D11017	WORD	Память для хранения названий рецептов. Задание 41. Символ 18
D11018	WORD	Память для хранения названий рецептов. Задание 41. Символ 19
D11019	WORD	Память для хранения названий рецептов. Задание 41. Символ 20
D11020	WORD	Память для хранения названий рецептов. Задание 41. Символ 21
D11021	WORD	Память для хранения названий рецептов. Задание 41. Символ 22
D11022	WORD	Память для хранения названий рецептов. Задание 41. Символ 23
D11023	WORD	Память для хранения названий рецептов. Задание 41. Символ 24
D11024	WORD	Память для хранения названий рецептов. Задание 41. Символ 25
D11025	WORD	Память для хранения названий рецептов. Задание 42. Символ 1
D11026	WORD	Память для хранения названий рецептов. Задание 42. Символ 2
D11027	WORD	Память для хранения названий рецептов. Задание 42. Символ 3
D11028	WORD	Память для хранения названий рецептов. Задание 42. Символ 4
D11029	WORD	Память для хранения названий рецептов. Задание 42. Символ 5
D11030	WORD	Память для хранения названий рецептов. Задание 42. Символ 6
D11031	WORD	Память для хранения названий рецептов. Задание 42. Символ 7
D11032	WORD	Память для хранения названий рецептов. Задание 42. Символ 8
D11033	WORD	Память для хранения названий рецептов. Задание 42. Символ 9
D11034	WORD	Память для хранения названий рецептов. Задание 42. Символ 10
D11035	WORD	Память для хранения названий рецептов. Задание 42. Символ 11
D11036	WORD	Память для хранения названий рецептов. Задание 42. Символ 12
D11037	WORD	Память для хранения названий рецептов. Задание 42. Символ 13
D11038	WORD	Память для хранения названий рецептов. Задание 42. Символ 14
D11039	WORD	Память для хранения названий рецептов. Задание 42. Символ 15
D11040	WORD	Память для хранения названий рецептов. Задание 42. Символ 16
D11041	WORD	Память для хранения названий рецептов. Задание 42. Символ 17
D11042	WORD	Память для хранения названий рецептов. Задание 42. Символ 18
D11043	WORD	Память для хранения названий рецептов. Задание 42. Символ 19
D11044	WORD	Память для хранения названий рецептов. Задание 42. Символ 20
D11045	WORD	Память для хранения названий рецептов. Задание 42. Символ 21
D11046	WORD	Память для хранения названий рецептов. Задание 42. Символ 22
D11047	WORD	Память для хранения названий рецептов. Задание 42. Символ 23
D11048	WORD	Память для хранения названий рецептов. Задание 42. Символ 24
D11049	WORD	Память для хранения названий рецептов. Задание 42. Символ 25
D11050	WORD	Память для хранения названий рецептов. Задание 43. Символ 1
D11051	WORD	Память для хранения названий рецептов. Задание 43. Символ 2
D11052	WORD	Память для хранения названий рецептов. Задание 43. Символ 3
D11053	WORD	Память для хранения названий рецептов. Задание 43. Символ 4
D11054	WORD	Память для хранения названий рецептов. Задание 43. Символ 5
D11055	WORD	Память для хранения названий рецептов. Задание 43. Символ 6
D11056	WORD	Память для хранения названий рецептов. Задание 43. Символ 7
D11057	WORD	Память для хранения названий рецептов. Задание 43. Символ 8
D11058	WORD	Память для хранения названий рецептов. Задание 43. Символ 9
D11059	WORD	Память для хранения названий рецептов. Задание 43. Символ 10
D11060	WORD	Память для хранения названий рецептов. Задание 43. Символ 11
D11061	WORD	Память для хранения названий рецептов. Задание 43. Символ 12
D11062	WORD	Память для хранения названий рецептов. Задание 43. Символ 13
D11063	WORD	Память для хранения названий рецептов. Задание 43. Символ 14
D11064	WORD	Память для хранения названий рецептов. Задание 43. Символ 15
D11065	WORD	Память для хранения названий рецептов. Задание 43. Символ 16
D11066	WORD	Память для хранения названий рецептов. Задание 43. Символ 17
D11067	WORD	Память для хранения названий рецептов. Задание 43. Символ 18
D11068	WORD	Память для хранения названий рецептов. Задание 43. Символ 19
D11069	WORD	Память для хранения названий рецептов. Задание 43. Символ 20
D11070	WORD	Память для хранения названий рецептов. Задание 43. Символ 21
D11071	WORD	Память для хранения названий рецептов. Задание 43. Символ 22
D11072	WORD	Память для хранения названий рецептов. Задание 43. Символ 23
D11073	WORD	Память для хранения названий рецептов. Задание 43. Символ 24
D11074	WORD	Память для хранения названий рецептов. Задание 43. Символ 25
D11075	WORD	Память для хранения названий рецептов. Задание 44. Символ 1
D11076	WORD	Память для хранения названий рецептов. Задание 44. Символ 2
D11077	WORD	Память для хранения названий рецептов. Задание 44. Символ 3
D11078	WORD	Память для хранения названий рецептов. Задание 44. Символ 4
D11079	WORD	Память для хранения названий рецептов. Задание 44. Символ 5
D11080	WORD	Память для хранения названий рецептов. Задание 44. Символ 6
D11081	WORD	Память для хранения названий рецептов. Задание 44. Символ 7
D11082	WORD	Память для хранения названий рецептов. Задание 44. Символ 8
D11083	WORD	Память для хранения названий рецептов. Задание 44. Символ 9
D11084	WORD	Память для хранения названий рецептов. Задание 44. Символ 10
D11085	WORD	Память для хранения названий рецептов. Задание 44. Символ 11
D11086	WORD	Память для хранения названий рецептов. Задание 44. Символ 12
D11087	WORD	Память для хранения названий рецептов. Задание 44. Символ 13
D11088	WORD	Память для хранения названий рецептов. Задание 44. Символ 14
D11089	WORD	Память для хранения названий рецептов. Задание 44. Символ 15
D11090	WORD	Память для хранения названий рецептов. Задание 44. Символ 16
D11091	WORD	Память для хранения названий рецептов. Задание 44. Символ 17
D11092	WORD	Память для хранения названий рецептов. Задание 44. Символ 18
D11093	WORD	Память для хранения названий рецептов. Задание 44. Символ 19
D11094	WORD	Память для хранения названий рецептов. Задание 44. Символ 20
D11095	WORD	Память для хранения названий рецептов. Задание 44. Символ 21
D11096	WORD	Память для хранения названий рецептов. Задание 44. Символ 22
D11097	WORD	Память для хранения названий рецептов. Задание 44. Символ 23
D11098	WORD	Память для хранения названий рецептов. Задание 44. Символ 24
D11099	WORD	Память для хранения названий рецептов. Задание 44. Символ 25
D11100	WORD	Память для хранения названий рецептов. Задание 45. Символ 1
D11101	WORD	Память для хранения названий рецептов. Задание 45. Символ 2
D11102	WORD	Память для хранения названий рецептов. Задание 45. Символ 3
D11103	WORD	Память для хранения названий рецептов. Задание 45. Символ 4
D11104	WORD	Память для хранения названий рецептов. Задание 45. Символ 5
D11105	WORD	Память для хранения названий рецептов. Задание 45. Символ 6
D11106	WORD	Память для хранения названий рецептов. Задание 45. Символ 7
D11107	WORD	Память для хранения названий рецептов. Задание 45. Символ 8
D11108	WORD	Память для хранения названий рецептов. Задание 45. Символ 9
D11109	WORD	Память для хранения названий рецептов. Задание 45. Символ 10
D11110	WORD	Память для хранения названий рецептов. Задание 45. Символ 11
D11111	WORD	Память для хранения названий рецептов. Задание 45. Символ 12
D11112	WORD	Память для хранения названий рецептов. Задание 45. Символ 13
D11113	WORD	Память для хранения названий рецептов. Задание 45. Символ 14
D11114	WORD	Память для хранения названий рецептов. Задание 45. Символ 15
D11115	WORD	Память для хранения названий рецептов. Задание 45. Символ 16
D11116	WORD	Память для хранения названий рецептов. Задание 45. Символ 17
D11117	WORD	Память для хранения названий рецептов. Задание 45. Символ 18
D11118	WORD	Память для хранения названий рецептов. Задание 45. Символ 19
D11119	WORD	Память для хранения названий рецептов. Задание 45. Символ 20
D11120	WORD	Память для хранения названий рецептов. Задание 45. Символ 21
D11121	WORD	Память для хранения названий рецептов. Задание 45. Символ 22
D11122	WORD	Память для хранения названий рецептов. Задание 45. Символ 23
D11123	WORD	Память для хранения названий рецептов. Задание 45. Символ 24
D11124	WORD	Память для хранения названий рецептов. Задание 45. Символ 25
D11125	WORD	Память для хранения названий рецептов. Задание 46. Символ 1
D11126	WORD	Память для хранения названий рецептов. Задание 46. Символ 2
D11127	WORD	Память для хранения названий рецептов. Задание 46. Символ 3
D11128	WORD	Память для хранения названий рецептов. Задание 46. Символ 4
D11129	WORD	Память для хранения названий рецептов. Задание 46. Символ 5
D11130	WORD	Память для хранения названий рецептов. Задание 46. Символ 6
D11131	WORD	Память для хранения названий рецептов. Задание 46. Символ 7
D11132	WORD	Память для хранения названий рецептов. Задание 46. Символ 8
D11133	WORD	Память для хранения названий рецептов. Задание 46. Символ 9
D11134	WORD	Память для хранения названий рецептов. Задание 46. Символ 10
D11135	WORD	Память для хранения названий рецептов. Задание 46. Символ 11
D11136	WORD	Память для хранения названий рецептов. Задание 46. Символ 12
D11137	WORD	Память для хранения названий рецептов. Задание 46. Символ 13
D11138	WORD	Память для хранения названий рецептов. Задание 46. Символ 14
D11139	WORD	Память для хранения названий рецептов. Задание 46. Символ 15
D11140	WORD	Память для хранения названий рецептов. Задание 46. Символ 16
D11141	WORD	Память для хранения названий рецептов. Задание 46. Символ 17
D11142	WORD	Память для хранения названий рецептов. Задание 46. Символ 18
D11143	WORD	Память для хранения названий рецептов. Задание 46. Символ 19
D11144	WORD	Память для хранения названий рецептов. Задание 46. Символ 20
D11145	WORD	Память для хранения названий рецептов. Задание 46. Символ 21
D11146	WORD	Память для хранения названий рецептов. Задание 46. Символ 22
D11147	WORD	Память для хранения названий рецептов. Задание 46. Символ 23
D11148	WORD	Память для хранения названий рецептов. Задание 46. Символ 24
D11149	WORD	Память для хранения названий рецептов. Задание 46. Символ 25
D11150	WORD	Память для хранения названий рецептов. Задание 47. Символ 1
D11151	WORD	Память для хранения названий рецептов. Задание 47. Символ 2
D11152	WORD	Память для хранения названий рецептов. Задание 47. Символ 3
D11153	WORD	Память для хранения названий рецептов. Задание 47. Символ 4
D11154	WORD	Память для хранения названий рецептов. Задание 47. Символ 5
D11155	WORD	Память для хранения названий рецептов. Задание 47. Символ 6
D11156	WORD	Память для хранения названий рецептов. Задание 47. Символ 7
D11157	WORD	Память для хранения названий рецептов. Задание 47. Символ 8
D11158	WORD	Память для хранения названий рецептов. Задание 47. Символ 9
D11159	WORD	Память для хранения названий рецептов. Задание 47. Символ 10
D11160	WORD	Память для хранения названий рецептов. Задание 47. Символ 11
D11161	WORD	Память для хранения названий рецептов. Задание 47. Символ 12
D11162	WORD	Память для хранения названий рецептов. Задание 47. Символ 13
D11163	WORD	Память для хранения названий рецептов. Задание 47. Символ 14
D11164	WORD	Память для хранения названий рецептов. Задание 47. Символ 15
D11165	WORD	Память для хранения названий рецептов. Задание 47. Символ 16
D11166	WORD	Память для хранения названий рецептов. Задание 47. Символ 17
D11167	WORD	Память для хранения названий рецептов. Задание 47. Символ 18
D11168	WORD	Память для хранения названий рецептов. Задание 47. Символ 19
D11169	WORD	Память для хранения названий рецептов. Задание 47. Символ 20
D11170	WORD	Память для хранения названий рецептов. Задание 47. Символ 21
D11171	WORD	Память для хранения названий рецептов. Задание 47. Символ 22
D11172	WORD	Память для хранения названий рецептов. Задание 47. Символ 23
D11173	WORD	Память для хранения названий рецептов. Задание 47. Символ 24
D11174	WORD	Память для хранения названий рецептов. Задание 47. Символ 25
D11175	WORD	Память для хранения названий рецептов. Задание 48. Символ 1
D11176	WORD	Память для хранения названий рецептов. Задание 48. Символ 2
D11177	WORD	Память для хранения названий рецептов. Задание 48. Символ 3
D11178	WORD	Память для хранения названий рецептов. Задание 48. Символ 4
D11179	WORD	Память для хранения названий рецептов. Задание 48. Символ 5
D11180	WORD	Память для хранения названий рецептов. Задание 48. Символ 6
D11181	WORD	Память для хранения названий рецептов. Задание 48. Символ 7
D11182	WORD	Память для хранения названий рецептов. Задание 48. Символ 8
D11183	WORD	Память для хранения названий рецептов. Задание 48. Символ 9
D11184	WORD	Память для хранения названий рецептов. Задание 48. Символ 10
D11185	WORD	Память для хранения названий рецептов. Задание 48. Символ 11
D11186	WORD	Память для хранения названий рецептов. Задание 48. Символ 12
D11187	WORD	Память для хранения названий рецептов. Задание 48. Символ 13
D11188	WORD	Память для хранения названий рецептов. Задание 48. Символ 14
D11189	WORD	Память для хранения названий рецептов. Задание 48. Символ 15
D11190	WORD	Память для хранения названий рецептов. Задание 48. Символ 16
D11191	WORD	Память для хранения названий рецептов. Задание 48. Символ 17
D11192	WORD	Память для хранения названий рецептов. Задание 48. Символ 18
D11193	WORD	Память для хранения названий рецептов. Задание 48. Символ 19
D11194	WORD	Память для хранения названий рецептов. Задание 48. Символ 20
D11195	WORD	Память для хранения названий рецептов. Задание 48. Символ 21
D11196	WORD	Память для хранения названий рецептов. Задание 48. Символ 22
D11197	WORD	Память для хранения названий рецептов. Задание 48. Символ 23
D11198	WORD	Память для хранения названий рецептов. Задание 48. Символ 24
D11199	WORD	Память для хранения названий рецептов. Задание 48. Символ 25
D11200	WORD	Память для хранения названий рецептов. Задание 49. Символ 1
D11201	WORD	Память для хранения названий рецептов. Задание 49. Символ 2
D11202	WORD	Память для хранения названий рецептов. Задание 49. Символ 3
D11203	WORD	Память для хранения названий рецептов. Задание 49. Символ 4
D11204	WORD	Память для хранения названий рецептов. Задание 49. Символ 5
D11205	WORD	Память для хранения названий рецептов. Задание 49. Символ 6
D11206	WORD	Память для хранения названий рецептов. Задание 49. Символ 7
D11207	WORD	Память для хранения названий рецептов. Задание 49. Символ 8
D11208	WORD	Память для хранения названий рецептов. Задание 49. Символ 9
D11209	WORD	Память для хранения названий рецептов. Задание 49. Символ 10
D11210	WORD	Память для хранения названий рецептов. Задание 49. Символ 11
D11211	WORD	Память для хранения названий рецептов. Задание 49. Символ 12
D11212	WORD	Память для хранения названий рецептов. Задание 49. Символ 13
D11213	WORD	Память для хранения названий рецептов. Задание 49. Символ 14
D11214	WORD	Память для хранения названий рецептов. Задание 49. Символ 15
D11215	WORD	Память для хранения названий рецептов. Задание 49. Символ 16
D11216	WORD	Память для хранения названий рецептов. Задание 49. Символ 17
D11217	WORD	Память для хранения названий рецептов. Задание 49. Символ 18
D11218	WORD	Память для хранения названий рецептов. Задание 49. Символ 19
D11219	WORD	Память для хранения названий рецептов. Задание 49. Символ 20
D11220	WORD	Память для хранения названий рецептов. Задание 49. Символ 21
D11221	WORD	Память для хранения названий рецептов. Задание 49. Символ 22
D11222	WORD	Память для хранения названий рецептов. Задание 49. Символ 23
D11223	WORD	Память для хранения названий рецептов. Задание 49. Символ 24
D11224	WORD	Память для хранения названий рецептов. Задание 49. Символ 25
D11225	WORD	Память для хранения названий рецептов. Задание 50. Символ 1
D11226	WORD	Память для хранения названий рецептов. Задание 50. Символ 2
D11227	WORD	Память для хранения названий рецептов. Задание 50. Символ 3
D11228	WORD	Память для хранения названий рецептов. Задание 50. Символ 4
D11229	WORD	Память для хранения названий рецептов. Задание 50. Символ 5
D11230	WORD	Память для хранения названий рецептов. Задание 50. Символ 6
D11231	WORD	Память для хранения названий рецептов. Задание 50. Символ 7
D11232	WORD	Память для хранения названий рецептов. Задание 50. Символ 8
D11233	WORD	Память для хранения названий рецептов. Задание 50. Символ 9
D11234	WORD	Память для хранения названий рецептов. Задание 50. Символ 10
D11235	WORD	Память для хранения названий рецептов. Задание 50. Символ 11
D11236	WORD	Память для хранения названий рецептов. Задание 50. Символ 12
D11237	WORD	Память для хранения названий рецептов. Задание 50. Символ 13
D11238	WORD	Память для хранения названий рецептов. Задание 50. Символ 14
D11239	WORD	Память для хранения названий рецептов. Задание 50. Символ 15
D11240	WORD	Память для хранения названий рецептов. Задание 50. Символ 16
D11241	WORD	Память для хранения названий рецептов. Задание 50. Символ 17
D11242	WORD	Память для хранения названий рецептов. Задание 50. Символ 18
D11243	WORD	Память для хранения названий рецептов. Задание 50. Символ 19
D11244	WORD	Память для хранения названий рецептов. Задание 50. Символ 20
D11245	WORD	Память для хранения названий рецептов. Задание 50. Символ 21
D11246	WORD	Память для хранения названий рецептов. Задание 50. Символ 22
D11247	WORD	Память для хранения названий рецептов. Задание 50. Символ 23
D11248	WORD	Память для хранения названий рецептов. Задание 50. Символ 24
D11249	WORD	Память для хранения названий рецептов. Задание 50. Символ 25
D11250	WORD	Память для хранения названий рецептов. Задание 51. Символ 1
D11251	WORD	Память для хранения названий рецептов. Задание 51. Символ 2
D11252	WORD	Память для хранения названий рецептов. Задание 51. Символ 3
D11253	WORD	Память для хранения названий рецептов. Задание 51. Символ 4
D11254	WORD	Память для хранения названий рецептов. Задание 51. Символ 5
D11255	WORD	Память для хранения названий рецептов. Задание 51. Символ 6
D11256	WORD	Память для хранения названий рецептов. Задание 51. Символ 7
D11257	WORD	Память для хранения названий рецептов. Задание 51. Символ 8
D11258	WORD	Память для хранения названий рецептов. Задание 51. Символ 9
D11259	WORD	Память для хранения названий рецептов. Задание 51. Символ 10
D11260	WORD	Память для хранения названий рецептов. Задание 51. Символ 11
D11261	WORD	Память для хранения названий рецептов. Задание 51. Символ 12
D11262	WORD	Память для хранения названий рецептов. Задание 51. Символ 13
D11263	WORD	Память для хранения названий рецептов. Задание 51. Символ 14
D11264	WORD	Память для хранения названий рецептов. Задание 51. Символ 15
D11265	WORD	Память для хранения названий рецептов. Задание 51. Символ 16
D11266	WORD	Память для хранения названий рецептов. Задание 51. Символ 17
D11267	WORD	Память для хранения названий рецептов. Задание 51. Символ 18
D11268	WORD	Память для хранения названий рецептов. Задание 51. Символ 19
D11269	WORD	Память для хранения названий рецептов. Задание 51. Символ 20
D11270	WORD	Память для хранения названий рецептов. Задание 51. Символ 21
D11271	WORD	Память для хранения названий рецептов. Задание 51. Символ 22
D11272	WORD	Память для хранения названий рецептов. Задание 51. Символ 23
D11273	WORD	Память для хранения названий рецептов. Задание 51. Символ 24
D11274	WORD	Память для хранения названий рецептов. Задание 51. Символ 25
D11275	WORD	Память для хранения названий рецептов. Задание 52. Символ 1
D11276	WORD	Память для хранения названий рецептов. Задание 52. Символ 2
D11277	WORD	Память для хранения названий рецептов. Задание 52. Символ 3
D11278	WORD	Память для хранения названий рецептов. Задание 52. Символ 4
D11279	WORD	Память для хранения названий рецептов. Задание 52. Символ 5
D11280	WORD	Память для хранения названий рецептов. Задание 52. Символ 6
D11281	WORD	Память для хранения названий рецептов. Задание 52. Символ 7
D11282	WORD	Память для хранения названий рецептов. Задание 52. Символ 8
D11283	WORD	Память для хранения названий рецептов. Задание 52. Символ 9
D11284	WORD	Память для хранения названий рецептов. Задание 52. Символ 10
D11285	WORD	Память для хранения названий рецептов. Задание 52. Символ 11
D11286	WORD	Память для хранения названий рецептов. Задание 52. Символ 12
D11287	WORD	Память для хранения названий рецептов. Задание 52. Символ 13
D11288	WORD	Память для хранения названий рецептов. Задание 52. Символ 14
D11289	WORD	Память для хранения названий рецептов. Задание 52. Символ 15
D11290	WORD	Память для хранения названий рецептов. Задание 52. Символ 16
D11291	WORD	Память для хранения названий рецептов. Задание 52. Символ 17
D11292	WORD	Память для хранения названий рецептов. Задание 52. Символ 18
D11293	WORD	Память для хранения названий рецептов. Задание 52. Символ 19
D11294	WORD	Память для хранения названий рецептов. Задание 52. Символ 20
D11295	WORD	Память для хранения названий рецептов. Задание 52. Символ 21
D11296	WORD	Память для хранения названий рецептов. Задание 52. Символ 22
D11297	WORD	Память для хранения названий рецептов. Задание 52. Символ 23
D11298	WORD	Память для хранения названий рецептов. Задание 52. Символ 24
D11299	WORD	Память для хранения названий рецептов. Задание 52. Символ 25
D11300	WORD	Память для хранения названий рецептов. Задание 53. Символ 1
D11301	WORD	Память для хранения названий рецептов. Задание 53. Символ 2
D11302	WORD	Память для хранения названий рецептов. Задание 53. Символ 3
D11303	WORD	Память для хранения названий рецептов. Задание 53. Символ 4
D11304	WORD	Память для хранения названий рецептов. Задание 53. Символ 5
D11305	WORD	Память для хранения названий рецептов. Задание 53. Символ 6
D11306	WORD	Память для хранения названий рецептов. Задание 53. Символ 7
D11307	WORD	Память для хранения названий рецептов. Задание 53. Символ 8
D11308	WORD	Память для хранения названий рецептов. Задание 53. Символ 9
D11309	WORD	Память для хранения названий рецептов. Задание 53. Символ 10
D11310	WORD	Память для хранения названий рецептов. Задание 53. Символ 11
D11311	WORD	Память для хранения названий рецептов. Задание 53. Символ 12
D11312	WORD	Память для хранения названий рецептов. Задание 53. Символ 13
D11313	WORD	Память для хранения названий рецептов. Задание 53. Символ 14
D11314	WORD	Память для хранения названий рецептов. Задание 53. Символ 15
D11315	WORD	Память для хранения названий рецептов. Задание 53. Символ 16
D11316	WORD	Память для хранения названий рецептов. Задание 53. Символ 17
D11317	WORD	Память для хранения названий рецептов. Задание 53. Символ 18
D11318	WORD	Память для хранения названий рецептов. Задание 53. Символ 19
D11319	WORD	Память для хранения названий рецептов. Задание 53. Символ 20
D11320	WORD	Память для хранения названий рецептов. Задание 53. Символ 21
D11321	WORD	Память для хранения названий рецептов. Задание 53. Символ 22
D11322	WORD	Память для хранения названий рецептов. Задание 53. Символ 23
D11323	WORD	Память для хранения названий рецептов. Задание 53. Символ 24
D11324	WORD	Память для хранения названий рецептов. Задание 53. Символ 25
D11325	WORD	Память для хранения названий рецептов. Задание 54. Символ 1
D11326	WORD	Память для хранения названий рецептов. Задание 54. Символ 2
D11327	WORD	Память для хранения названий рецептов. Задание 54. Символ 3
D11328	WORD	Память для хранения названий рецептов. Задание 54. Символ 4
D11329	WORD	Память для хранения названий рецептов. Задание 54. Символ 5
D11330	WORD	Память для хранения названий рецептов. Задание 54. Символ 6
D11331	WORD	Память для хранения названий рецептов. Задание 54. Символ 7
D11332	WORD	Память для хранения названий рецептов. Задание 54. Символ 8
D11333	WORD	Память для хранения названий рецептов. Задание 54. Символ 9
D11334	WORD	Память для хранения названий рецептов. Задание 54. Символ 10
D11335	WORD	Память для хранения названий рецептов. Задание 54. Символ 11
D11336	WORD	Память для хранения названий рецептов. Задание 54. Символ 12
D11337	WORD	Память для хранения названий рецептов. Задание 54. Символ 13
D11338	WORD	Память для хранения названий рецептов. Задание 54. Символ 14
D11339	WORD	Память для хранения названий рецептов. Задание 54. Символ 15
D11340	WORD	Память для хранения названий рецептов. Задание 54. Символ 16
D11341	WORD	Память для хранения названий рецептов. Задание 54. Символ 17
D11342	WORD	Память для хранения названий рецептов. Задание 54. Символ 18
D11343	WORD	Память для хранения названий рецептов. Задание 54. Символ 19
D11344	WORD	Память для хранения названий рецептов. Задание 54. Символ 20
D11345	WORD	Память для хранения названий рецептов. Задание 54. Символ 21
D11346	WORD	Память для хранения названий рецептов. Задание 54. Символ 22
D11347	WORD	Память для хранения названий рецептов. Задание 54. Символ 23
D11348	WORD	Память для хранения названий рецептов. Задание 54. Символ 24
D11349	WORD	Память для хранения названий рецептов. Задание 54. Символ 25
D11350	WORD	Память для хранения названий рецептов. Задание 55. Символ 1
D11351	WORD	Память для хранения названий рецептов. Задание 55. Символ 2
D11352	WORD	Память для хранения названий рецептов. Задание 55. Символ 3
D11353	WORD	Память для хранения названий рецептов. Задание 55. Символ 4
D11354	WORD	Память для хранения названий рецептов. Задание 55. Символ 5
D11355	WORD	Память для хранения названий рецептов. Задание 55. Символ 6
D11356	WORD	Память для хранения названий рецептов. Задание 55. Символ 7
D11357	WORD	Память для хранения названий рецептов. Задание 55. Символ 8
D11358	WORD	Память для хранения названий рецептов. Задание 55. Символ 9
D11359	WORD	Память для хранения названий рецептов. Задание 55. Символ 10
D11360	WORD	Память для хранения названий рецептов. Задание 55. Символ 11
D11361	WORD	Память для хранения названий рецептов. Задание 55. Символ 12
D11362	WORD	Память для хранения названий рецептов. Задание 55. Символ 13
D11363	WORD	Память для хранения названий рецептов. Задание 55. Символ 14
D11364	WORD	Память для хранения названий рецептов. Задание 55. Символ 15
D11365	WORD	Память для хранения названий рецептов. Задание 55. Символ 16
D11366	WORD	Память для хранения названий рецептов. Задание 55. Символ 17
D11367	WORD	Память для хранения названий рецептов. Задание 55. Символ 18
D11368	WORD	Память для хранения названий рецептов. Задание 55. Символ 19
D11369	WORD	Память для хранения названий рецептов. Задание 55. Символ 20
D11370	WORD	Память для хранения названий рецептов. Задание 55. Символ 21
D11371	WORD	Память для хранения названий рецептов. Задание 55. Символ 22
D11372	WORD	Память для хранения названий рецептов. Задание 55. Символ 23
D11373	WORD	Память для хранения названий рецептов. Задание 55. Символ 24
D11374	WORD	Память для хранения названий рецептов. Задание 55. Символ 25
D11375	WORD	Память для хранения названий рецептов. Задание 56. Символ 1
D11376	WORD	Память для хранения названий рецептов. Задание 56. Символ 2
D11377	WORD	Память для хранения названий рецептов. Задание 56. Символ 3
D11378	WORD	Память для хранения названий рецептов. Задание 56. Символ 4
D11379	WORD	Память для хранения названий рецептов. Задание 56. Символ 5
D11380	WORD	Память для хранения названий рецептов. Задание 56. Символ 6
D11381	WORD	Память для хранения названий рецептов. Задание 56. Символ 7
D11382	WORD	Память для хранения названий рецептов. Задание 56. Символ 8
D11383	WORD	Память для хранения названий рецептов. Задание 56. Символ 9
D11384	WORD	Память для хранения названий рецептов. Задание 56. Символ 10
D11385	WORD	Память для хранения названий рецептов. Задание 56. Символ 11
D11386	WORD	Память для хранения названий рецептов. Задание 56. Символ 12
D11387	WORD	Память для хранения названий рецептов. Задание 56. Символ 13
D11388	WORD	Память для хранения названий рецептов. Задание 56. Символ 14
D11389	WORD	Память для хранения названий рецептов. Задание 56. Символ 15
D11390	WORD	Память для хранения названий рецептов. Задание 56. Символ 16
D11391	WORD	Память для хранения названий рецептов. Задание 56. Символ 17
D11392	WORD	Память для хранения названий рецептов. Задание 56. Символ 18
D11393	WORD	Память для хранения названий рецептов. Задание 56. Символ 19
D11394	WORD	Память для хранения названий рецептов. Задание 56. Символ 20
D11395	WORD	Память для хранения названий рецептов. Задание 56. Символ 21
D11396	WORD	Память для хранения названий рецептов. Задание 56. Символ 22
D11397	WORD	Память для хранения названий рецептов. Задание 56. Символ 23
D11398	WORD	Память для хранения названий рецептов. Задание 56. Символ 24
D11399	WORD	Память для хранения названий рецептов. Задание 56. Символ 25
D11400	WORD	Память для хранения названий рецептов. Задание 57. Символ 1
D11401	WORD	Память для хранения названий рецептов. Задание 57. Символ 2
D11402	WORD	Память для хранения названий рецептов. Задание 57. Символ 3
D11403	WORD	Память для хранения названий рецептов. Задание 57. Символ 4
D11404	WORD	Память для хранения названий рецептов. Задание 57. Символ 5
D11405	WORD	Память для хранения названий рецептов. Задание 57. Символ 6
D11406	WORD	Память для хранения названий рецептов. Задание 57. Символ 7
D11407	WORD	Память для хранения названий рецептов. Задание 57. Символ 8
D11408	WORD	Память для хранения названий рецептов. Задание 57. Символ 9
D11409	WORD	Память для хранения названий рецептов. Задание 57. Символ 10
D11410	WORD	Память для хранения названий рецептов. Задание 57. Символ 11
D11411	WORD	Память для хранения названий рецептов. Задание 57. Символ 12
D11412	WORD	Память для хранения названий рецептов. Задание 57. Символ 13
D11413	WORD	Память для хранения названий рецептов. Задание 57. Символ 14
D11414	WORD	Память для хранения названий рецептов. Задание 57. Символ 15
D11415	WORD	Память для хранения названий рецептов. Задание 57. Символ 16
D11416	WORD	Память для хранения названий рецептов. Задание 57. Символ 17
D11417	WORD	Память для хранения названий рецептов. Задание 57. Символ 18
D11418	WORD	Память для хранения названий рецептов. Задание 57. Символ 19
D11419	WORD	Память для хранения названий рецептов. Задание 57. Символ 20
D11420	WORD	Память для хранения названий рецептов. Задание 57. Символ 21
D11421	WORD	Память для хранения названий рецептов. Задание 57. Символ 22
D11422	WORD	Память для хранения названий рецептов. Задание 57. Символ 23
D11423	WORD	Память для хранения названий рецептов. Задание 57. Символ 24
D11424	WORD	Память для хранения названий рецептов. Задание 57. Символ 25
D11425	WORD	Память для хранения названий рецептов. Задание 58. Символ 1
D11426	WORD	Память для хранения названий рецептов. Задание 58. Символ 2
D11427	WORD	Память для хранения названий рецептов. Задание 58. Символ 3
D11428	WORD	Память для хранения названий рецептов. Задание 58. Символ 4
D11429	WORD	Память для хранения названий рецептов. Задание 58. Символ 5
D11430	WORD	Память для хранения названий рецептов. Задание 58. Символ 6
D11431	WORD	Память для хранения названий рецептов. Задание 58. Символ 7
D11432	WORD	Память для хранения названий рецептов. Задание 58. Символ 8
D11433	WORD	Память для хранения названий рецептов. Задание 58. Символ 9
D11434	WORD	Память для хранения названий рецептов. Задание 58. Символ 10
D11435	WORD	Память для хранения названий рецептов. Задание 58. Символ 11
D11436	WORD	Память для хранения названий рецептов. Задание 58. Символ 12
D11437	WORD	Память для хранения названий рецептов. Задание 58. Символ 13
D11438	WORD	Память для хранения названий рецептов. Задание 58. Символ 14
D11439	WORD	Память для хранения названий рецептов. Задание 58. Символ 15
D11440	WORD	Память для хранения названий рецептов. Задание 58. Символ 16
D11441	WORD	Память для хранения названий рецептов. Задание 58. Символ 17
D11442	WORD	Память для хранения названий рецептов. Задание 58. Символ 18
D11443	WORD	Память для хранения названий рецептов. Задание 58. Символ 19
D11444	WORD	Память для хранения названий рецептов. Задание 58. Символ 20
D11445	WORD	Память для хранения названий рецептов. Задание 58. Символ 21
D11446	WORD	Память для хранения названий рецептов. Задание 58. Символ 22
D11447	WORD	Память для хранения названий рецептов. Задание 58. Символ 23
D11448	WORD	Память для хранения названий рецептов. Задание 58. Символ 24
D11449	WORD	Память для хранения названий рецептов. Задание 58. Символ 25
D11450	WORD	Память для хранения названий рецептов. Задание 59. Символ 1
D11451	WORD	Память для хранения названий рецептов. Задание 59. Символ 2
D11452	WORD	Память для хранения названий рецептов. Задание 59. Символ 3
D11453	WORD	Память для хранения названий рецептов. Задание 59. Символ 4
D11454	WORD	Память для хранения названий рецептов. Задание 59. Символ 5
D11455	WORD	Память для хранения названий рецептов. Задание 59. Символ 6
D11456	WORD	Память для хранения названий рецептов. Задание 59. Символ 7
D11457	WORD	Память для хранения названий рецептов. Задание 59. Символ 8
D11458	WORD	Память для хранения названий рецептов. Задание 59. Символ 9
D11459	WORD	Память для хранения названий рецептов. Задание 59. Символ 10
D11460	WORD	Память для хранения названий рецептов. Задание 59. Символ 11
D11461	WORD	Память для хранения названий рецептов. Задание 59. Символ 12
D11462	WORD	Память для хранения названий рецептов. Задание 59. Символ 13
D11463	WORD	Память для хранения названий рецептов. Задание 59. Символ 14
D11464	WORD	Память для хранения названий рецептов. Задание 59. Символ 15
D11465	WORD	Память для хранения названий рецептов. Задание 59. Символ 16
D11466	WORD	Память для хранения названий рецептов. Задание 59. Символ 17
D11467	WORD	Память для хранения названий рецептов. Задание 59. Символ 18
D11468	WORD	Память для хранения названий рецептов. Задание 59. Символ 19
D11469	WORD	Память для хранения названий рецептов. Задание 59. Символ 20
D11470	WORD	Память для хранения названий рецептов. Задание 59. Символ 21
D11471	WORD	Память для хранения названий рецептов. Задание 59. Символ 22
D11472	WORD	Память для хранения названий рецептов. Задание 59. Символ 23
D11473	WORD	Память для хранения названий рецептов. Задание 59. Символ 24
D11474	WORD	Память для хранения названий рецептов. Задание 59. Символ 25
D11475	WORD	Память для хранения названий рецептов. Задание 60. Символ 1
D11476	WORD	Память для хранения названий рецептов. Задание 60. Символ 2
D11477	WORD	Память для хранения названий рецептов. Задание 60. Символ 3
D11478	WORD	Память для хранения названий рецептов. Задание 60. Символ 4
D11479	WORD	Память для хранения названий рецептов. Задание 60. Символ 5
D11480	WORD	Память для хранения названий рецептов. Задание 60. Символ 6
D11481	WORD	Память для хранения названий рецептов. Задание 60. Символ 7
D11482	WORD	Память для хранения названий рецептов. Задание 60. Символ 8
D11483	WORD	Память для хранения названий рецептов. Задание 60. Символ 9
D11484	WORD	Память для хранения названий рецептов. Задание 60. Символ 10
D11485	WORD	Память для хранения названий рецептов. Задание 60. Символ 11
D11486	WORD	Память для хранения названий рецептов. Задание 60. Символ 12
D11487	WORD	Память для хранения названий рецептов. Задание 60. Символ 13
D11488	WORD	Память для хранения названий рецептов. Задание 60. Символ 14
D11489	WORD	Память для хранения названий рецептов. Задание 60. Символ 15
D11490	WORD	Память для хранения названий рецептов. Задание 60. Символ 16
D11491	WORD	Память для хранения названий рецептов. Задание 60. Символ 17
D11492	WORD	Память для хранения названий рецептов. Задание 60. Символ 18
D11493	WORD	Память для хранения названий рецептов. Задание 60. Символ 19
D11494	WORD	Память для хранения названий рецептов. Задание 60. Символ 20
D11495	WORD	Память для хранения названий рецептов. Задание 60. Символ 21
D11496	WORD	Память для хранения названий рецептов. Задание 60. Символ 22
D11497	WORD	Память для хранения названий рецептов. Задание 60. Символ 23
D11498	WORD	Память для хранения названий рецептов. Задание 60. Символ 24
D11499	WORD	Память для хранения названий рецептов. Задание 60. Символ 25
D11500	WORD	Память для хранения названий рецептов. Задание 58. Символ 19
D11501	WORD	Память для хранения названий рецептов. Задание 58. Символ 20
D11502	WORD	Память для хранения названий рецептов. Задание 58. Символ 21
D11503	WORD	Память для хранения названий рецептов. Задание 58. Символ 22
D11504	WORD	Память для хранения названий рецептов. Задание 58. Символ 23
D11505	WORD	Память для хранения названий рецептов. Задание 58. Символ 24
D11506	WORD	Память для хранения названий рецептов. Задание 58. Символ 25
D11507	WORD	Память для хранения названий рецептов. Задание 59. Символ 0
D11508	WORD	Память для хранения названий рецептов. Задание 59. Символ 1
D11509	WORD	Память для хранения названий рецептов. Задание 59. Символ 2
D11510	WORD	Память для хранения названий рецептов. Задание 59. Символ 3
D11511	WORD	Память для хранения названий рецептов. Задание 59. Символ 4
D00171	WORD	Предыдущая выбранная пластина 
T0012	BIT/WORD	100MS Время на смену номера блока и номера рецепта
T0015	BIT/WORD	100MS Таймер сброса команды загрузки данных
T0016	BIT/WORD	100MS Таймер сброса команды сохранения данных
T0017	BIT/WORD	100MS Время на смену номера блока и номера рецепта
T0018	BIT/WORD	100MS Время на смену номера блока и номера рецепта
D00168	WORD	Смещение номера ред. пластины на 100
D00173	WORD	Номер редактируемой пластины -101
T0019	BIT/WORD	100MS Время на смену номера блока и номера рецепта
D00180	WORD	Последняя загруженная пластина
D00175	WORD	Оффсет строки для выбранного номера пластины
D00176	WORD	MULNULL
D00177	WORD	MULNULL
D00178	WORD	MULNULL
D00319.0	BIT	Смещение чётного ряда (0)
D00320.0	BIT	Смещение первого ряда относительно нуля Х (0)
M00145	BIT	Кнопка сохранения пластины в базу данных
M00151	BIT	Флаг сохранения пластины
Z00004	WORD	Смещение редактируемого имени пластины
M00149	BIT	Требуется загрузка пластины при редактировании
T0034	BIT/WORD	100MS Таймер на подготовку данных перед загрузкой
D00174	WORD	Номер редактируемой пластины -1
M0014A	BIT	Флаг загрузки пластины при редактировании
M0014B	BIT	Загрузка при первом открытии рецепта пластин
D00190	WORD	Выбранная пластина -1
M0014E	BIT	Флаг загрузки задания при запуске цикла
M0014F	BIT	Требуется загрузка задания при запуске цикла
M00152	BIT	Загрузка один раз при запуске цикла
T0036	BIT/WORD	100MS Таймер на подготовку данных перед загрузкой
D00321.0	BIT	Смещение первого ряда относительно нуля Y (0)
P11110	BIT	Таймер открытия патрона 2 (0)
D10960	WORD	Память для хранения названий рецептов. Задание 39. Символ 11
D10961	WORD	Память для хранения названий рецептов. Задание 39. Символ 12
D10962	WORD	Память для хранения названий рецептов. Задание 39. Символ 13
D10963	WORD	Память для хранения названий рецептов. Задание 39. Символ 14
D10964	WORD	Память для хранения названий рецептов. Задание 39. Символ 15
D10965	WORD	Память для хранения названий рецептов. Задание 39. Символ 16
D10966	WORD	Память для хранения названий рецептов. Задание 39. Символ 17
D10967	WORD	Память для хранения названий рецептов. Задание 39. Символ 18
D10968	WORD	Память для хранения названий рецептов. Задание 39. Символ 19
D10969	WORD	Память для хранения названий рецептов. Задание 39. Символ 20
D10970	WORD	Память для хранения названий рецептов. Задание 39. Символ 21
D10971	WORD	Память для хранения названий рецептов. Задание 39. Символ 22
D10972	WORD	Память для хранения названий рецептов. Задание 39. Символ 23
D10973	WORD	Память для хранения названий рецептов. Задание 39. Символ 24
D10974	WORD	Память для хранения названий рецептов. Задание 39. Символ 25
D10975	WORD	Память для хранения названий рецептов. Задание 40. Символ 1
D10976	WORD	Память для хранения названий рецептов. Задание 40. Символ 2
D10977	WORD	Память для хранения названий рецептов. Задание 40. Символ 3
D10978	WORD	Память для хранения названий рецептов. Задание 40. Символ 4
D10979	WORD	Память для хранения названий рецептов. Задание 40. Символ 5
D10980	WORD	Память для хранения названий рецептов. Задание 40. Символ 6
D10981	WORD	Память для хранения названий рецептов. Задание 40. Символ 7
D10982	WORD	Память для хранения названий рецептов. Задание 40. Символ 8
D10983	WORD	Память для хранения названий рецептов. Задание 40. Символ 9
D10984	WORD	Память для хранения названий рецептов. Задание 40. Символ 10
D10985	WORD	Память для хранения названий рецептов. Задание 40. Символ 11
D10986	WORD	Память для хранения названий рецептов. Задание 40. Символ 12
D10987	WORD	Память для хранения названий рецептов. Задание 40. Символ 13
D10988	WORD	Память для хранения названий рецептов. Задание 40. Символ 14
D10989	WORD	Память для хранения названий рецептов. Задание 40. Символ 15
D10990	WORD	Память для хранения названий рецептов. Задание 40. Символ 16
D10991	WORD	Память для хранения названий рецептов. Задание 40. Символ 17
D10992	WORD	Память для хранения названий рецептов. Задание 40. Символ 18
D10993	WORD	Память для хранения названий рецептов. Задание 40. Символ 19
D10994	WORD	Память для хранения названий рецептов. Задание 40. Символ 20
D10995	WORD	Память для хранения названий рецептов. Задание 40. Символ 21
D10996	WORD	Память для хранения названий рецептов. Задание 40. Символ 22
D10997	WORD	Память для хранения названий рецептов. Задание 40. Символ 23
D10998	WORD	Память для хранения названий рецептов. Задание 40. Символ 24
D10999	WORD	Память для хранения названий рецептов. Задание 40. Символ 25
D11512	WORD	Память для хранения названий рецептов. Задание 59. Символ 5
D11513	WORD	Память для хранения названий рецептов. Задание 59. Символ 6
D11514	WORD	Память для хранения названий рецептов. Задание 59. Символ 7
D11515	WORD	Память для хранения названий рецептов. Задание 59. Символ 8
D11516	WORD	Память для хранения названий рецептов. Задание 59. Символ 9
D11517	WORD	Память для хранения названий рецептов. Задание 59. Символ 10
D11518	WORD	Память для хранения названий рецептов. Задание 59. Символ 11
D11519	WORD	Память для хранения названий рецептов. Задание 59. Символ 12
D11520	WORD	Память для хранения названий рецептов. Задание 59. Символ 13
D11521	WORD	Память для хранения названий рецептов. Задание 59. Символ 14
D11522	WORD	Память для хранения названий рецептов. Задание 59. Символ 15
D11523	WORD	Память для хранения названий рецептов. Задание 59. Символ 16
D11524	WORD	Память для хранения названий рецептов. Задание 59. Символ 17
D11525	WORD	Память для хранения названий рецептов. Задание 59. Символ 18
D11526	WORD	Память для хранения названий рецептов. Задание 59. Символ 19
D11527	WORD	Память для хранения названий рецептов. Задание 59. Символ 20
D11528	WORD	Память для хранения названий рецептов. Задание 59. Символ 21
D11529	WORD	Память для хранения названий рецептов. Задание 59. Символ 22
D11530	WORD	Память для хранения названий рецептов. Задание 59. Символ 23
D11531	WORD	Память для хранения названий рецептов. Задание 59. Символ 24
D11532	WORD	Память для хранения названий рецептов. Задание 59. Символ 25
D11533	WORD	Память для хранения названий рецептов. Задание 60. Символ 0
D11534	WORD	Память для хранения названий рецептов. Задание 60. Символ 1
D11535	WORD	Память для хранения названий рецептов. Задание 60. Символ 2
D11536	WORD	Память для хранения названий рецептов. Задание 60. Символ 3
D11537	WORD	Память для хранения названий рецептов. Задание 60. Символ 4
D11538	WORD	Память для хранения названий рецептов. Задание 60. Символ 5
D11539	WORD	Память для хранения названий рецептов. Задание 60. Символ 6
D11540	WORD	Память для хранения названий рецептов. Задание 60. Символ 7
D11541	WORD	Память для хранения названий рецептов. Задание 60. Символ 8
D11542	WORD	Память для хранения названий рецептов. Задание 60. Символ 9
D11543	WORD	Память для хранения названий рецептов. Задание 60. Символ 10
D11544	WORD	Память для хранения названий рецептов. Задание 60. Символ 11
D11545	WORD	Память для хранения названий рецептов. Задание 60. Символ 12
D11546	WORD	Память для хранения названий рецептов. Задание 60. Символ 13
D11547	WORD	Память для хранения названий рецептов. Задание 60. Символ 14
D11548	WORD	Память для хранения названий рецептов. Задание 60. Символ 15
D11549	WORD	Память для хранения названий рецептов. Задание 60. Символ 16
D11550	WORD	Память для хранения названий рецептов. Задание 60. Символ 17
D11551	WORD	Память для хранения названий рецептов. Задание 60. Символ 18
D11552	WORD	Память для хранения названий рецептов. Задание 60. Символ 19
D11553	WORD	Память для хранения названий рецептов. Задание 60. Символ 20
D11554	WORD	Память для хранения названий рецептов. Задание 60. Символ 21
D11555	WORD	Память для хранения названий рецептов. Задание 60. Символ 22
D11556	WORD	Память для хранения названий рецептов. Задание 60. Символ 23
D11557	WORD	Память для хранения названий рецептов. Задание 60. Символ 24
D11558	WORD	Память для хранения названий рецептов. Задание 60. Символ 25
D00250	WORD	Пароль от уровня 1
D00256	WORD	Пароль от уровня 2
D12001	WORD	Редактируемое имя задания. Символ 2
D12002	WORD	Редактируемое имя задания. Символ 3
D12003	WORD	Редактируемое имя задания. Символ 4
D12004	WORD	Редактируемое имя задания. Символ 5
D12005	WORD	Редактируемое имя задания. Символ 6
D12006	WORD	Редактируемое имя задания. Символ 7
D12007	WORD	Редактируемое имя задания. Символ 8
D12008	WORD	Редактируемое имя задания. Символ 9
D12009	WORD	Редактируемое имя задания. Символ 10
D12010	WORD	Редактируемое имя задания. Символ 11
D12011	WORD	Редактируемое имя задания. Символ 12
D12012	WORD	Редактируемое имя задания. Символ 13
D12013	WORD	Редактируемое имя задания. Символ 14
D12014	WORD	Редактируемое имя задания. Символ 15
D12015	WORD	Редактируемое имя задания. Символ 16
D12016	WORD	Редактируемое имя задания. Символ 17
D12017	WORD	Редактируемое имя задания. Символ 18
D12018	WORD	Редактируемое имя задания. Символ 19
D12019	WORD	Редактируемое имя задания. Символ 20
D12020	WORD	Редактируемое имя задания. Символ 21
D12021	WORD	Редактируемое имя задания. Символ 22
D12022	WORD	Редактируемое имя задания. Символ 23
D12023	WORD	Редактируемое имя задания. Символ 24
D12024	WORD	Редактируемое имя задания. Символ 25
P11310	BIT	Инверсия захвата 1
P11311	BIT	Инверсия захвата 2
P11312	BIT	Требуется запуск программы на станке
P11313	BIT	Требуется обдув перед установкой детали
P11314	BIT	Требуется обдув после забора детали
P11315	BIT	Забираем готовую деталь из патрона 1
P11316	BIT	Забираем готовую деталь из патрона 2
P11317	BIT	Сначала открываем захват, а потом закрываем патрон
P11318	BIT	Сначала закрываем патрон, а потом открываем захват
D00331	WORD	Резерв
D00332.0	BIT	Инверсия захвата 1
P10018	BIT	Захват 2 открыт (датчик)
P10019	BIT	Захват 2 открыт (команда)
P1001A	BIT	Захват 2 закрыт (команда)
P1001B	BIT	Ошибка открытия захвата 2 (при наличии датчика)
P1001C	BIT	Усилие на захвате 2 (датчик)
P10050	BIT	Код ошибки на роботе (0)
P10051	BIT	Код ошибки на роботе (1)
P10052	BIT	Код ошибки на роботе (2)
P10053	BIT	Код ошибки на роботе (3)
P10054	BIT	Код ошибки на роботе (4)
P10055	BIT	Код ошибки на роботе (5)
P10056	BIT	Код ошибки на роботе (6)
P10057	BIT	Код ошибки на роботе (7)
P10058	BIT	Код ошибки на роботе (8)
P10059	BIT	Код ошибки на роботе (9)
P1005A	BIT	Код ошибки на роботе (10)
P1005B	BIT	Код ошибки на роботе (11)
P1005C	BIT	Код ошибки на роботе (12)
P1005D	BIT	Код ошибки на роботе (13)
P1005E	BIT	Код ошибки на роботе (14)
P1005F	BIT	Код ошибки на роботе (15)
P10061	BIT	Номер захвата 1 (1)
P10062	BIT	Номер захвата 1 (2)
P10063	BIT	Номер захвата 1 (3)
P10064	BIT	Номер захвата 1 (4)
P10065	BIT	Номер захвата 1 (5)
P10066	BIT	Номер захвата 1 (6)
P10067	BIT	Номер захвата 1 (7)
P10069	BIT	Номер захвата 2 (1)
P1006A	BIT	Номер захвата 2 (2)
P1006B	BIT	Номер захвата 2 (3)
P1006C	BIT	Номер захвата 2 (4)
P1006D	BIT	Номер захвата 2 (5)
P1006E	BIT	Номер захвата 2 (6)
P1006F	BIT	Номер захвата 2 (7)
P10071	BIT	Номер патрона 1 (1)
P10072	BIT	Номер патрона 1 (2)
P10073	BIT	Номер патрона 1 (3)
P10074	BIT	Номер патрона 1 (4)
P10075	BIT	Номер патрона 1 (5)
P10076	BIT	Номер патрона 1 (6)
P10077	BIT	Номер патрона 1 (7)
P10079	BIT	Номер патрона 2 / станции перехвата (1)
P1007A	BIT	Номер патрона 2 / станции перехвата (2)
P1007B	BIT	Номер патрона 2 / станции перехвата (3)
P1007C	BIT	Номер патрона 2 / станции перехвата (4)
P1007D	BIT	Номер патрона 2 / станции перехвата (5)
P1007E	BIT	Номер патрона 2 / станции перехвата (6)
P1007F	BIT	Номер патрона 2 / станции перехвата (7)
P10081	BIT	Обработано деталей (1)
P10082	BIT	Обработано деталей (2)
P10083	BIT	Обработано деталей (3)
P10084	BIT	Обработано деталей (4)
P10085	BIT	Обработано деталей (5)
P10086	BIT	Обработано деталей (6)
P10087	BIT	Обработано деталей (7)
P10089	BIT	Следующая деталь (1)
P1008A	BIT	Следующая деталь (2)
P1008B	BIT	Следующая деталь (3)
P1008C	BIT	Следующая деталь (4)
P1008D	BIT	Следующая деталь (5)
P1008E	BIT	Следующая деталь (6)
P1008F	BIT	Следующая деталь (7)
P11018	BIT	Открыть захват 2 с HMI
P11019	BIT	Закрыть захват 2 с HMI
P11051	BIT	Скорость робота (1)
P11052	BIT	Скорость робота (2)
P11053	BIT	Скорость робота (3)
P11054	BIT	Скорость робота (4)
P11055	BIT	Скорость робота (5)
P11056	BIT	Скорость робота (6)
P11057	BIT	Скорость робота (7)
P11061	BIT	Скорость поиска (1)
P11062	BIT	Скорость поиска (2)
P11063	BIT	Скорость поиска (3)
P11064	BIT	Скорость поиска (4)
P11065	BIT	Скорость поиска (5)
P11066	BIT	Скорость поиска (6)
P11067	BIT	Скорость поиска (7)
P11069	BIT	Скорость обдува (1)
P1106A	BIT	Скорость обдува (2)
P1106B	BIT	Скорость обдува (3)
P1106C	BIT	Скорость обдува (4)
P1106D	BIT	Скорость обдува (5)
P1106E	BIT	Скорость обдува (6)
P1106F	BIT	Скорость обдува (7)
P11071	BIT	Overshoot при поиске (1)
P11072	BIT	Overshoot при поиске (2)
P11073	BIT	Overshoot при поиске (3)
P11081	BIT	Таймер открытия захвата 1 (1)
P11082	BIT	Таймер открытия захвата 1 (2)
P11083	BIT	Таймер открытия захвата 1 (3)
P11084	BIT	Таймер открытия захвата 1 (4)
P11085	BIT	Таймер открытия захвата 1 (5)
P11086	BIT	Таймер открытия захвата 1 (6)
P11087	BIT	Таймер открытия захвата 1 (7)
P11089	BIT	Таймер закрытия захвата 1 (1)
P1108A	BIT	Таймер закрытия захвата 1 (2)
P1108B	BIT	Таймер закрытия захвата 1 (3)
P1108C	BIT	Таймер закрытия захвата 1 (4)
P1108D	BIT	Таймер закрытия захвата 1 (5)
P1108E	BIT	Таймер закрытия захвата 1 (6)
P1108F	BIT	Таймер закрытия захвата 1 (7)
P11091	BIT	Таймер открытия захвата 2 (1)
P11092	BIT	Таймер открытия захвата 2 (2)
P11093	BIT	Таймер открытия захвата 2 (3)
P11094	BIT	Таймер открытия захвата 2 (4)
P11095	BIT	Таймер открытия захвата 2 (5)
P11096	BIT	Таймер открытия захвата 2 (6)
P11097	BIT	Таймер открытия захвата 2 (7)
P11099	BIT	Таймер закрытия захвата 2 (1)
P1109A	BIT	Таймер закрытия захвата 2 (2)
P1109B	BIT	Таймер закрытия захвата 2 (3)
P1109C	BIT	Таймер закрытия захвата 2 (4)
P1109D	BIT	Таймер закрытия захвата 2 (5)
P1109E	BIT	Таймер закрытия захвата 2 (6)
P1109F	BIT	Таймер закрытия захвата 2 (7)
P11102	BIT	Таймер открытия патрона 1 (2)
P11103	BIT	Таймер открытия патрона 1 (3)
P11104	BIT	Таймер открытия патрона 1 (4)
P11105	BIT	Таймер открытия патрона 1 (5)
P11106	BIT	Таймер открытия патрона 1 (6)
P11107	BIT	Таймер открытия патрона 1 (7)
P11109	BIT	Таймер закрытия патрона 1 (1)
P1110A	BIT	Таймер закрытия патрона 1 (2)
P1110B	BIT	Таймер закрытия патрона 1 (3)
P1110C	BIT	Таймер закрытия патрона 1 (4)
P1110D	BIT	Таймер закрытия патрона 1 (5)
P1110E	BIT	Таймер закрытия патрона 1 (6)
P1110F	BIT	Таймер закрытия патрона 1 (7)
P11112	BIT	Таймер открытия патрона 2 (2)
P11113	BIT	Таймер открытия патрона 2 (3)
P11114	BIT	Таймер открытия патрона 2 (4)
P11115	BIT	Таймер открытия патрона 2 (5)
P11116	BIT	Таймер открытия патрона 2 (6)
P11117	BIT	Таймер открытия патрона 2 (7)
P11119	BIT	Таймер закрытия патрона 2 (1)
P1111A	BIT	Таймер закрытия патрона 2 (2)
P1111B	BIT	Таймер закрытия патрона 2 (3)
P1111C	BIT	Таймер закрытия патрона 2 (4)
P1111D	BIT	Таймер закрытия патрона 2 (5)
P1111E	BIT	Таймер закрытия патрона 2 (6)
P1111F	BIT	Таймер закрытия патрона 2 (7)
P11161	BIT	Длина заготовки (1)
P11162	BIT	Длина заготовки (2)
P11163	BIT	Длина заготовки (3)
P11164	BIT	Длина заготовки (4)
P11165	BIT	Длина заготовки (5)
P11166	BIT	Длина заготовки (6)
P11167	BIT	Длина заготовки (7)
P11169	BIT	Длина обработанной с одной стороны детали (1)
P1116A	BIT	Длина обработанной с одной стороны детали (2)
P1116B	BIT	Длина обработанной с одной стороны детали (3)
P1116C	BIT	Длина обработанной с одной стороны детали (4)
P1116D	BIT	Длина обработанной с одной стороны детали (5)
P1116E	BIT	Длина обработанной с одной стороны детали (6)
P1116F	BIT	Длина обработанной с одной стороны детали (7)
P11171	BIT	Длина готовой детали (1)
P11172	BIT	Длина готовой детали (2)
P11173	BIT	Длина готовой детали (3)
P11174	BIT	Длина готовой детали (4)
P11175	BIT	Длина готовой детали (5)
P11176	BIT	Длина готовой детали (6)
P11177	BIT	Длина готовой детали (7)
P11179	BIT	Полная длина кулачков на захвате 1 (1)
P1117A	BIT	Полная длина кулачков на захвате 1 (2)
P1117B	BIT	Полная длина кулачков на захвате 1 (3)
P1117C	BIT	Полная длина кулачков на захвате 1 (4)
P1117D	BIT	Полная длина кулачков на захвате 1 (5)
P1117E	BIT	Полная длина кулачков на захвате 1 (6)
P1117F	BIT	Полная длина кулачков на захвате 1 (7)
P11181	BIT	Тело кулачков на захвате 1 (1)
P11182	BIT	Тело кулачков на захвате 1 (2)
P11183	BIT	Тело кулачков на захвате 1 (3)
P11184	BIT	Тело кулачков на захвате 1 (4)
P11185	BIT	Тело кулачков на захвате 1 (5)
P11186	BIT	Тело кулачков на захвате 1 (6)
P11187	BIT	Тело кулачков на захвате 1 (7)
P11189	BIT	Полная длина кулачков на захвате 2 (1)
P1118A	BIT	Полная длина кулачков на захвате 2 (2)
P1118B	BIT	Полная длина кулачков на захвате 2 (3)
P1118C	BIT	Полная длина кулачков на захвате 2 (4)
P1118D	BIT	Полная длина кулачков на захвате 2 (5)
P1118E	BIT	Полная длина кулачков на захвате 2 (6)
P1118F	BIT	Полная длина кулачков на захвате 2 (7)
P11191	BIT	Тело кулачков на захвате 2 (1)
P11192	BIT	Тело кулачков на захвате 2 (2)
P11193	BIT	Тело кулачков на захвате 2 (3)
P11194	BIT	Тело кулачков на захвате 2 (4)
P11195	BIT	Тело кулачков на захвате 2 (5)
P11196	BIT	Тело кулачков на захвате 2 (6)
P11197	BIT	Тело кулачков на захвате 2 (7)
P11199	BIT	Полная длина кулачков в патроне 1 (1)
P1119A	BIT	Полная длина кулачков в патроне 1 (2)
P1119B	BIT	Полная длина кулачков в патроне 1 (3)
P1119C	BIT	Полная длина кулачков в патроне 1 (4)
P1119D	BIT	Полная длина кулачков в патроне 1 (5)
P1119E	BIT	Полная длина кулачков в патроне 1 (6)
P1119F	BIT	Полная длина кулачков в патроне 1 (7)
P11201	BIT	Тело кулачков в патроне 1 (1)
P11202	BIT	Тело кулачков в патроне 1 (2)
P11203	BIT	Тело кулачков в патроне 1 (3)
P11204	BIT	Тело кулачков в патроне 1 (4)
P11205	BIT	Тело кулачков в патроне 1 (5)
P11206	BIT	Тело кулачков в патроне 1 (6)
P11207	BIT	Тело кулачков в патроне 1 (7)
P11209	BIT	Полная длина кулачков в патроне 2/ ст.перехвата (1)
P1120A	BIT	Полная длина кулачков в патроне 2/ ст.перехвата (2)
P1120B	BIT	Полная длина кулачков в патроне 2/ ст.перехвата (3)
P1120C	BIT	Полная длина кулачков в патроне 2/ ст.перехвата (4)
P1120D	BIT	Полная длина кулачков в патроне 2/ ст.перехвата (5)
P1120E	BIT	Полная длина кулачков в патроне 2/ ст.перехвата (6)
P1120F	BIT	Полная длина кулачков в патроне 2/ ст.перехвата (7)
P11211	BIT	Тело кулачков в патроне 2/ ст.перехвата  (1)
P11212	BIT	Тело кулачков в патроне 2/ ст.перехвата  (2)
P11213	BIT	Тело кулачков в патроне 2/ ст.перехвата  (3)
P11214	BIT	Тело кулачков в патроне 2/ ст.перехвата  (4)
P11215	BIT	Тело кулачков в патроне 2/ ст.перехвата  (5)
P11216	BIT	Тело кулачков в патроне 2/ ст.перехвата  (6)
P11217	BIT	Тело кулачков в патроне 2/ ст.перехвата  (7)
P11219	BIT	Количество рядов на пластине (1)
P1121A	BIT	Количество рядов на пластине (2)
P1121B	BIT	Количество рядов на пластине (3)
P1121D	BIT	Количество ячеек в нечётных рядах (1)
P1121E	BIT	Количество ячеек в нечётных рядах (2)
P1121F	BIT	Количество ячеек в нечётных рядах (3)
P11221	BIT	Количество ячеек в чётных рядах (1)
P11222	BIT	Количество ячеек в чётных рядах (2)
P11223	BIT	Количество ячеек в чётных рядах (3)
P11230	BIT	Расстояние между ячейками (0)
P11231	BIT	Расстояние между ячейками (1)
P11232	BIT	Расстояние между ячейками (2)
P11233	BIT	Расстояние между ячейками (3)
P11234	BIT	Расстояние между ячейками (4)
P11235	BIT	Расстояние между ячейками (5)
P11236	BIT	Расстояние между ячейками (6)
P11237	BIT	Расстояние между ячейками (7)
P11238	BIT	Расстояние между ячейками (8)
P11239	BIT	Расстояние между ячейками (9)
P1123A	BIT	Расстояние между ячейками (10)
P1123B	BIT	Расстояние между ячейками (11)
P1123C	BIT	Расстояние между ячейками (12)
P1123D	BIT	Расстояние между ячейками (13)
P1123E	BIT	Расстояние между ячейками (14)
P1123F	BIT	Расстояние между ячейками (15)
P11240	BIT	Расстояние между рядами (0)
P11241	BIT	Расстояние между рядами (1)
P11242	BIT	Расстояние между рядами (2)
P11243	BIT	Расстояние между рядами (3)
P11244	BIT	Расстояние между рядами (4)
P11245	BIT	Расстояние между рядами (5)
P11246	BIT	Расстояние между рядами (6)
P11247	BIT	Расстояние между рядами (7)
P11248	BIT	Расстояние между рядами (8)
P11249	BIT	Расстояние между рядами (9)
P1124A	BIT	Расстояние между рядами (10)
P1124B	BIT	Расстояние между рядами (11)
P1124C	BIT	Расстояние между рядами (12)
P1124D	BIT	Расстояние между рядами (13)
P1124E	BIT	Расстояние между рядами (14)
P1124F	BIT	Расстояние между рядами (15)
P11250	BIT	Смещение чётного ряда (0)
P11251	BIT	Смещение чётного ряда (1)
P11252	BIT	Смещение чётного ряда (2)
P11253	BIT	Смещение чётного ряда (3)
P11254	BIT	Смещение чётного ряда (4)
P11255	BIT	Смещение чётного ряда (5)
P11256	BIT	Смещение чётного ряда (6)
P11257	BIT	Смещение чётного ряда (7)
P11258	BIT	Смещение чётного ряда (8)
P11259	BIT	Смещение чётного ряда (9)
P1125A	BIT	Смещение чётного ряда (10)
P1125B	BIT	Смещение чётного ряда (11)
P1125C	BIT	Смещение чётного ряда (12)
P1125D	BIT	Смещение чётного ряда (13)
P1125E	BIT	Смещение чётного ряда (14)
P1125F	BIT	Смещение чётного ряда (15)
P11260	BIT	Смещение первого ряда относительно нуля Х (0)
P11261	BIT	Смещение первого ряда относительно нуля Х (1)
P11262	BIT	Смещение первого ряда относительно нуля Х (2)
P11263	BIT	Смещение первого ряда относительно нуля Х (3)
P11264	BIT	Смещение первого ряда относительно нуля Х (4)
P11265	BIT	Смещение первого ряда относительно нуля Х (5)
P11266	BIT	Смещение первого ряда относительно нуля Х (6)
P11267	BIT	Смещение первого ряда относительно нуля Х (7)
P11268	BIT	Смещение первого ряда относительно нуля Х (8)
P11269	BIT	Смещение первого ряда относительно нуля Х (9)
P1126A	BIT	Смещение первого ряда относительно нуля Х (10)
P1126B	BIT	Смещение первого ряда относительно нуля Х (11)
P1126C	BIT	Смещение первого ряда относительно нуля Х (12)
P1126D	BIT	Смещение первого ряда относительно нуля Х (13)
P1126E	BIT	Смещение первого ряда относительно нуля Х (14)
P1126F	BIT	Смещение первого ряда относительно нуля Х (15)
P11270	BIT	Смещение первого ряда относительно нуля Y (0)
P11271	BIT	Смещение первого ряда относительно нуля Y (1)
P11272	BIT	Смещение первого ряда относительно нуля Y (2)
P11273	BIT	Смещение первого ряда относительно нуля Y (3)
P11274	BIT	Смещение первого ряда относительно нуля Y (4)
P11275	BIT	Смещение первого ряда относительно нуля Y (5)
P11276	BIT	Смещение первого ряда относительно нуля Y (6)
P11277	BIT	Смещение первого ряда относительно нуля Y (7)
P11278	BIT	Смещение первого ряда относительно нуля Y (8)
P11279	BIT	Смещение первого ряда относительно нуля Y (9)
P1127A	BIT	Смещение первого ряда относительно нуля Y (10)
P1127B	BIT	Смещение первого ряда относительно нуля Y (11)
P1127C	BIT	Смещение первого ряда относительно нуля Y (12)
P1127D	BIT	Смещение первого ряда относительно нуля Y (13)
P1127E	BIT	Смещение первого ряда относительно нуля Y (14)
P1127F	BIT	Смещение первого ряда относительно нуля Y (15)
P11281	BIT	Номер программы на станке (1)
P11282	BIT	Номер программы на станке (2)
P11283	BIT	Номер программы на станке (3)
P11284	BIT	Номер программы на станке (4)
P11285	BIT	Номер программы на станке (5)
P11286	BIT	Номер программы на станке (6)
P11287	BIT	Номер программы на станке (7)
P11289	BIT	Номер кастомной программы перехвата 1 (1)
P1128A	BIT	Номер кастомной программы перехвата 1 (2)
P1128B	BIT	Номер кастомной программы перехвата 1 (3)
P1128C	BIT	Номер кастомной программы перехвата 1 (4)
P1128D	BIT	Номер кастомной программы перехвата 1 (5)
P1128E	BIT	Номер кастомной программы перехвата 1 (6)
P1128F	BIT	Номер кастомной программы перехвата 1 (7)
P11291	BIT	Номер программы обдува 1 (1)
P11292	BIT	Номер программы обдува 1 (2)
P11293	BIT	Номер программы обдува 1 (3)
P11294	BIT	Номер программы обдува 1 (4)
P11295	BIT	Номер программы обдува 1 (5)
P11296	BIT	Номер программы обдува 1 (6)
P11297	BIT	Номер программы обдува 1 (7)
P11299	BIT	Номер программы обдува 2 (1)
P1129A	BIT	Номер программы обдува 2 (2)
P1129B	BIT	Номер программы обдува 2 (3)
P1129C	BIT	Номер программы обдува 2 (4)
P1129D	BIT	Номер программы обдува 2 (5)
P1129E	BIT	Номер программы обдува 2 (6)
P1129F	BIT	Номер программы обдува 2 (7)
P11301	BIT	Загружено ячеек (1)
P11302	BIT	Загружено ячеек (2)
P11303	BIT	Загружено ячеек (3)
P11304	BIT	Загружено ячеек (4)
P11305	BIT	Загружено ячеек (5)
P11306	BIT	Загружено ячеек (6)
P11307	BIT	Загружено ячеек (7)
P11308	BIT	Загружено ячеек (8)
P11319	BIT	Перехват внутри станка
P1131A	BIT	Внешняя станция перехвата
P1006	WORD	Номер захвата 1 (0)
P1007	WORD	Номер патрона 1 (0)
P1008	WORD	Обработано деталей (0)
P1105	WORD	Скорость робота (0)
P1106	WORD	Скорость поиска (0)
P1107	WORD	Overshoot при поиске (0)
P1108	WORD	Таймер открытия захвата 1 (0)
P1109	WORD	Таймер открытия захвата 2 (0)
P1111	WORD	Таймер открытия патрона 2 (0)
P1116	WORD	Длина заготовки (0)
P1117	WORD	Длина готовой детали (0)
P1118	WORD	Тело кулачков на захвате 1 (0)
P1119	WORD	Тело кулачков на захвате 2 (0)
P1120	WORD	Тело кулачков в патроне 1 (0)
P1121	WORD	Тело кулачков в патроне 2/ ст.перехвата  (0)
P1122	WORD	Количество ячеек в чётных рядах (0)
P1128	WORD	Номер программы на станке (0)
P1129	WORD	Номер программы обдува 1 (0)
P1130	WORD	Загружено ячеек (0)
D00000.0	BIT	Фиксированное число 0 (0)
D00001.0	BIT	Фиксированное число 1 (0)
D00002.0	BIT	Фиксированное число 2 (0)
D00003.0	BIT	Фиксированное число 3 (0)
D00004.0	BIT	Фиксированное число 4 (0)
D00005.0	BIT	Фиксированное число 5 (0)
D00006.0	BIT	Фиксированное число 6 (0)
D00007.0	BIT	Фиксированное число 7 (0)
D00008.0	BIT	Фиксированное число 8 (0)
D00009.0	BIT	Фиксированное число 9 (0)
D00010.0	BIT	Фиксированное число 10 (0)
D00011.0	BIT	Фиксированное число 11 (0)
D00012.0	BIT	Фиксированное число 12 (0)
D00013.0	BIT	Фиксированное число 13 (0)
D00014.0	BIT	Фиксированное число 14 (0)
D00015.0	BIT	Фиксированное число 15 (0)
D00016.0	BIT	Фиксированное число 16 (0)
D00017.0	BIT	Фиксированное число 17 (0)
D00018.0	BIT	Фиксированное число 18 (0)
D00019.0	BIT	Фиксированное число 19 (0)
D00020.0	BIT	Фиксированное число 20 (0)
D00021.0	BIT	Фиксированное число 21 (0)
D00022.0	BIT	Фиксированное число 22 (0)
D00023.0	BIT	Фиксированное число 23 (0)
D00024.0	BIT	Фиксированное число 24 (0)
D00025.0	BIT	Фиксированное число 25 (0)
D00026.0	BIT	Фиксированное число 26 (0)
D00027.0	BIT	Фиксированное число 27 (0)
D00028.0	BIT	Фиксированное число 28 (0)
D00029.0	BIT	Фиксированное число 29 (0)
D00030.0	BIT	Фиксированное число 30 (0)
D00031.0	BIT	Фиксированное число 31 (0)
D00032.0	BIT	Фиксированное число 32 (0)
D00033.0	BIT	Фиксированное число 33 (0)
D00034.0	BIT	Фиксированное число 34 (0)
D00035.0	BIT	Фиксированное число 35 (0)
D00036.0	BIT	Фиксированное число 36 (0)
D00037.0	BIT	Фиксированное число 37 (0)
D00038.0	BIT	Фиксированное число 38 (0)
D00039.0	BIT	Фиксированное число 39 (0)
D00040.0	BIT	Фиксированное число 40 (0)
D00041.0	BIT	Фиксированное число 41 (0)
D00042.0	BIT	Фиксированное число 42 (0)
D00043.0	BIT	Фиксированное число 43 (0)
D00044.0	BIT	Фиксированное число 44 (0)
D00045.0	BIT	Фиксированное число 45 (0)
D00046.0	BIT	Фиксированное число 46 (0)
D00047.0	BIT	Фиксированное число 47 (0)
D00048.0	BIT	Фиксированное число 48 (0)
D00049.0	BIT	Фиксированное число 49 (0)
D00050.0	BIT	Фиксированное число 50 (0)
D00051.0	BIT	Фиксированное число 51 (0)
D00052.0	BIT	Фиксированное число 52 (0)
D00053.0	BIT	Фиксированное число 53 (0)
D00054.0	BIT	Фиксированное число 54 (0)
D00055.0	BIT	Фиксированное число 55 (0)
D00056.0	BIT	Фиксированное число 56 (0)
D00057.0	BIT	Фиксированное число 57 (0)
D00058.0	BIT	Фиксированное число 58 (0)
D00059.0	BIT	Фиксированное число 59 (0)
D00060.0	BIT	Фиксированное число 60 (0)
D00061.0	BIT	Фиксированное число 61 (0)
D00062.0	BIT	Фиксированное число 62 (0)
D00063.0	BIT	Фиксированное число 63 (0)
D00064.0	BIT	Фиксированное число 64 (0)
D00065.0	BIT	Фиксированное число 65 (0)
D00066.0	BIT	Фиксированное число 66 (0)
D00067.0	BIT	Фиксированное число 67 (0)
D00068.0	BIT	Фиксированное число 68 (0)
D00069.0	BIT	Фиксированное число 69 (0)
D00070.0	BIT	Фиксированное число 70 (0)
D00071.0	BIT	Фиксированное число 71 (0)
D00072.0	BIT	Фиксированное число 72 (0)
D00073.0	BIT	Фиксированное число 73 (0)
D00074.0	BIT	Фиксированное число 74 (0)
D00075.0	BIT	Фиксированное число 75 (0)
D00076.0	BIT	Фиксированное число 76 (0)
D00077.0	BIT	Фиксированное число 77 (0)
D00078.0	BIT	Фиксированное число 78 (0)
D00079.0	BIT	Фиксированное число 79 (0)
D00080.0	BIT	Фиксированное число 80 (0)
D00081.0	BIT	Фиксированное число 81 (0)
D00082.0	BIT	Фиксированное число 82 (0)
D00083.0	BIT	Фиксированное число 83 (0)
D00084.0	BIT	Фиксированное число 84 (0)
D00085.0	BIT	Фиксированное число 85 (0)
D00086.0	BIT	Фиксированное число 86 (0)
D00087.0	BIT	Фиксированное число 87 (0)
D00088.0	BIT	Фиксированное число 88 (0)
D00089.0	BIT	Фиксированное число 89 (0)
D00090.0	BIT	Фиксированное число 90 (0)
D00091.0	BIT	Фиксированное число 91 (0)
D00092.0	BIT	Фиксированное число 92 (0)
D00093.0	BIT	Фиксированное число 93 (0)
D00094.0	BIT	Фиксированное число 94 (0)
D00095.0	BIT	Фиксированное число 95 (0)
D00096.0	BIT	Фиксированное число 96 (0)
D00097.0	BIT	Фиксированное число 97 (0)
D00098.0	BIT	Фиксированное число 98 (0)
D00099.0	BIT	Фиксированное число 99 (0)
D00100.0	BIT	Фиксированное число 100 (0)
D00101.0	BIT	Фиксированное число 101 (0)
D00102.0	BIT	Фиксированное число 102 (0)
D00103.0	BIT	Фиксированное число 103 (0)
D00104.0	BIT	Фиксированное число 104 (0)
D00105.0	BIT	Фиксированное число 105 (0)
D00106.0	BIT	Фиксированное число 106 (0)
D00107.0	BIT	Фиксированное число 107 (0)
D00108.0	BIT	Фиксированное число 108 (0)
D00109.0	BIT	Фиксированное число 109 (0)
D00110.0	BIT	Фиксированное число 110 (0)
D00111.0	BIT	Фиксированное число 111 (0)
D00112.0	BIT	Фиксированное число 112 (0)
D00113.0	BIT	Фиксированное число 113 (0)
D00114.0	BIT	Фиксированное число 114 (0)
D00115.0	BIT	Фиксированное число 115 (0)
D00116.0	BIT	Фиксированное число 116 (0)
D00117.0	BIT	Фиксированное число 117 (0)
D00118.0	BIT	Фиксированное число 118 (0)
D00119.0	BIT	Фиксированное число 119 (0)
D00120.0	BIT	Фиксированное число 120 (0)
D00121.0	BIT	Фиксированное число 121 (0)
D00122.0	BIT	Фиксированное число 122 (0)
D00123.0	BIT	Фиксированное число 123 (0)
D00124.0	BIT	Фиксированное число 124 (0)
D00125.0	BIT	Фиксированное число 125 (0)
D00126.0	BIT	Фиксированное число 126 (0)
D00127.0	BIT	Фиксированное число 127 (0)
D00128.0	BIT	Фиксированное число 128 (0)
D00131.0	BIT	HMI Время, в течении которого разблокирована полка после нажатия кнопки (0)
D00132.0	BIT	HMI Количество деталей на полке 1 (0)
D00133.0	BIT	HMI Количество деталей на полке 2 (0)
D00134.0	BIT	HMI Количество деталей на полке 3 (0)
D00135.0	BIT	HMI Количество деталей на полке 4 (0)
D00140.0	BIT	Выбранный номер задания (0)
D00141.0	BIT	Выбранный номер задания - 1 (0)
D00142.0	BIT	Оффсет строки для выбранного номера названия (0)
D00143.0	BIT	MULNULL (0)
D00144.0	BIT	MULNULL (0)
D00145.0	BIT	MULNULL (0)
D00146.0	BIT	Счётчик страницы заданий (0)
D00147.0	BIT	Оффсет номера страницы списка заданий (0)
D00148.0	BIT	MULNULL (0)
D00149.0	BIT	MULNULL (0)
D00150.0	BIT	MULNULL (0)
D00151.0	BIT	Оффсет строки страницы списка заданий (0)
D00152.0	BIT	MULNULL (0)
D00153.0	BIT	MULNULL (0)
D00154.0	BIT	MULNULL (0)
D00155.0	BIT	Номер кнопки на странице списка заданий (0)
D00156.0	BIT	Номер редактируемого задания (0)
D00157.0	BIT	Счётчик страницы пластин (0)
D00158.0	BIT	Оффсет номера страницы списка пластин (0)
D00159.0	BIT	MULNULL (0)
D00160.0	BIT	MULNULL (0)
D00161.0	BIT	MULNULL (0)
D00162.0	BIT	Оффсет строки страницы списка пластин (0)
D00163.0	BIT	MULNULL (0)
D00164.0	BIT	MULNULL (0)
D00165.0	BIT	MULNULL (0)
D00166.0	BIT	Номер кнопки на странице списка пластин (0)
D00167.0	BIT	Номер редактируемой пластины (0)
D00168.0	BIT	Смещение номера ред. пластины на 100 (0)
D00170.0	BIT	Предыдущее выбранное задание (0)
D00171.0	BIT	Предыдущая выбранная пластина  (0)
D00172.0	BIT	Номер редактируемого задания -1 (0)
D00173.0	BIT	Номер редактируемой пластины -101 (0)
D00174.0	BIT	Номер редактируемой пластины -1 (0)
D00175.0	BIT	Оффсет строки для выбранного номера пластины (0)
D00176.0	BIT	MULNULL (0)
D00177.0	BIT	MULNULL (0)
D00178.0	BIT	MULNULL (0)
D00180.0	BIT	Последняя загруженная пластина (0)
D00190.0	BIT	Выбранная пластина -1 (0)
D00199.0	BIT	Номер страницы HMI (0)
D00200.0	BIT	Код ошибки работы с базой данных (0)
D00201.0	BIT	Выбор типа рецепта (пластины/задания) (0)
D00202.0	BIT	Выбор блока рецепта (0)
D00203.0	BIT	Выбор номера файла (для EFR) (0)
D00250.0	BIT	Пароль от уровня 1 (0)
D00256.0	BIT	Пароль от уровня 2 (0)
D00300.0	BIT	Длина заготовки (0)
D00301.0	BIT	Диаметр заготоки (0)
D00302.0	BIT	Длина обработанной с одной стороны детали (0)
D00303.0	BIT	Диаметр обработанной с одной стороны детали (0)
D00304.0	BIT	Длина готовой детали (0)
D00305.0	BIT	Диаметр готовой детали (0)
D00306.0	BIT	Полная длина кулачков на захвате 1 (0)
D00307.0	BIT	Тело кулачков на захвате 1 (0)
D00308.0	BIT	Полная длина кулачков на захвате 2 (0)
D00309.0	BIT	Тело кулачков на захвате 2 (0)
D00310.0	BIT	Полная длина кулачков в патроне 1 (0)
D00311.0	BIT	Тело кулачков в патроне 1 (0)
D00312.0	BIT	Полная длина кулачков в патроне 2/ ст.перехвата (0)
D00313.0	BIT	Тело кулачков в патроне 2/ ст.перехвата (0)
D00317.0	BIT	Расстояние между ячейками (0)
D00318.0	BIT	Расстояние между рядами (0)
D00326.0	BIT	Резерв (0)
D00327.0	BIT	Резерв (0)
D00328.0	BIT	Резерв (0)
D00329.0	BIT	Резерв (0)
D00330.0	BIT	Резерв (0)
D00331.0	BIT	Резерв (0)
D00332.1	BIT	Инверсия захвата 2
D00332.3	BIT	Требуется обдув перед установкой детали
D00332.4	BIT	Требуется обдув после забора детали
D00332.9	BIT	Перехват внутри станка
D00332.A	BIT	Внешняя станция перехвата
D00230	WORD	Состояние захвата 1
D00231	WORD	Состояние захвата 2
D00232	WORD	Состояние патрона 1
D00233	WORD	Состояние патрона 2
D00234	WORD	Обработано деталей
D00414	WORD	Для робота: Количество рядов на пластине
D00415	WORD	Для робота: Количество ячеек в нечётных рядах
D00416	WORD	Для робота: Количество ячеек в чётных рядах
D00417	WORD	Для робота: Расстояние между ячейками
D00418	WORD	Для робота: Расстояние между рядами
D00419	WORD	Для робота: Смещение чётного ряда
D00420	WORD	Для робота: Смещение первого ряда относительно нуля Х
D00421	WORD	Для робота: Смещение первого ряда относительно нуля Y
D00422	WORD	Для робота: Номер программы на станке
D00423	WORD	Для робота: Номер кастомной программы перехвата
D00424	WORD	Для робота: Номер кастомной программы обдува перед установкой
D00425	WORD	Для робота: Номер кастомной программы обдува после установки
D00426	WORD	Для робота: Резерв
D00427	WORD	Для робота: Резерв
D00428	WORD	Для робота: Резерв
D00429	WORD	Для робота: Резерв
D00430	WORD	Для робота: Резерв
D00431	WORD	Для робота: Резерв
D00401.0	BIT	Для робота: Диаметр заготоки
D00403.0	BIT	Для робота: Диаметр обработанной с одной стороны детали
D00405.0	BIT	Для робота: Диаметр готовой детали
D00414.0	BIT	Для робота: Количество рядов на пластине
D00415.0	BIT	Для робота: Количество ячеек в нечётных рядах
D00416.0	BIT	Для робота: Количество ячеек в чётных рядах
D00417.0	BIT	Для робота: Расстояние между ячейками
D00418.0	BIT	Для робота: Расстояние между рядами
D00419.0	BIT	Для робота: Смещение чётного ряда
D00420.0	BIT	Для робота: Смещение первого ряда относительно нуля Х
D00421.0	BIT	Для робота: Смещение первого ряда относительно нуля Y
D00422.0	BIT	Для робота: Номер программы на станке
D00423.0	BIT	Для робота: Номер кастомной программы перехвата
D00424.0	BIT	Для робота: Номер кастомной программы обдува перед установкой
D00425.0	BIT	Для робота: Номер кастомной программы обдува после установки
D00426.0	BIT	Для робота: Резерв
D00427.0	BIT	Для робота: Резерв
D00428.0	BIT	Для робота: Резерв
D00429.0	BIT	Для робота: Резерв
D00430.0	BIT	Для робота: Резерв
D00431.0	BIT	Для робота: Резерв
P10090	BIT	Состояние захвата 1: пусто
P10091	BIT	Состояние захвата 1: заготовка
P10092	BIT	Состояние захвата 1: промежуток
P10093	BIT	Состояние захвата 1: деталь
P10094	BIT	Состояние захвата 2: пусто
P10095	BIT	Состояние захвата 2: заготовка
P10096	BIT	Состояние захвата 2: промежуток
P10097	BIT	Состояние захвата 2: деталь
P10098	BIT	Состояние патрона 1: пусто
P10099	BIT	Состояние патрона 1: заготовка
P1009A	BIT	Состояние патрона 1: промежуток
P1009B	BIT	Состояние патрона 1: деталь
P1009C	BIT	Состояние патрона 2: пусто
P1009D	BIT	Состояние патрона 2: заготовка
P1009E	BIT	Состояние патрона 2: промежуток
P1009F	BIT	Состояние патрона 2: деталь
// PLC CNCRemoteIO
// module base 0 slot 0: Input/Output Module:XBE-DR16A (DC 24V Input, Relay Output, 16 Contacts)
// module base 0 slot 1: Input/Output Module:XBE-DR16A (DC 24V Input, Relay Output, 16 Contacts)